(* CODESYS project escasa.project

Project tree, tasks and I/O mapping:
  Device : CODESYS Control Win V3, 3S - Smart Software Solutions GmbH, order no. 305021, version 3.5.10.30
    application Application
      libraries: Standard, * (System)
      task MainTask (cyclic, interval t#20ms, priority 1) calls PLC_PRG
      task VISU_TASK (cyclic, interval 100 ms, priority 31) calls VisuElems.Visu_Prg
      program PLC_PRG [ST]
      visualisation Visualization
  text list GlobalTextList
*)

// Device/Application/PLC_PRG
PROGRAM PLC_PRG
VAR
	green: BOOL := FALSE;
	yellow: BOOL := FALSE;
	red: BOOL := FALSE;
	onoff: BOOL;
	scelta: INT;
	
		
	
END_VAR

IF onoff = TRUE THEN	
	CASE scelta OF
	1: green := TRUE; red := FALSE; yellow := FALSE;
	2: green := FALSE; yellow := TRUE; red := FALSE;
	3: yellow := FALSE; red := TRUE; green := FALSE;
	ELSE 
	red := TRUE; green := TRUE; yellow := TRUE;
	END_CASE;
	
END_IF

END_PROGRAM

// Device/Application/Visualization
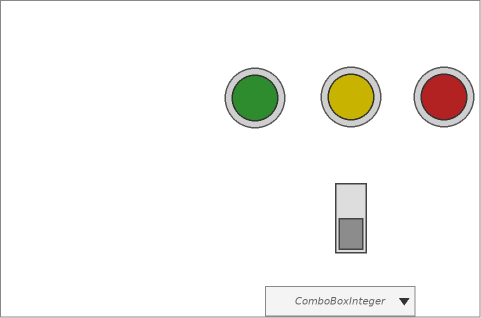
VISUALIZATION Visualization  // 481x318
    Lamp1 (409,62 70x70), variable: PLC_PRG.red, style: Lamp-Lamp1-Red
    Lamp1 (316,62 70x70), variable: PLC_PRG.yellow, style: Lamp-Lamp1-Yellow
    Lamp1 (220,63 70x70), variable: PLC_PRG.green, style: Lamp-Lamp1-Green
    DipSwitch (316,183 70x70), variable: PLC_PRG.onoff, behaviour: TOGGLE, style: Switch-DipSwitch-Gray
    ComboBoxInteger (265,286 150x30), variable: PLC_PRG.scelta
END_VISUALIZATION
